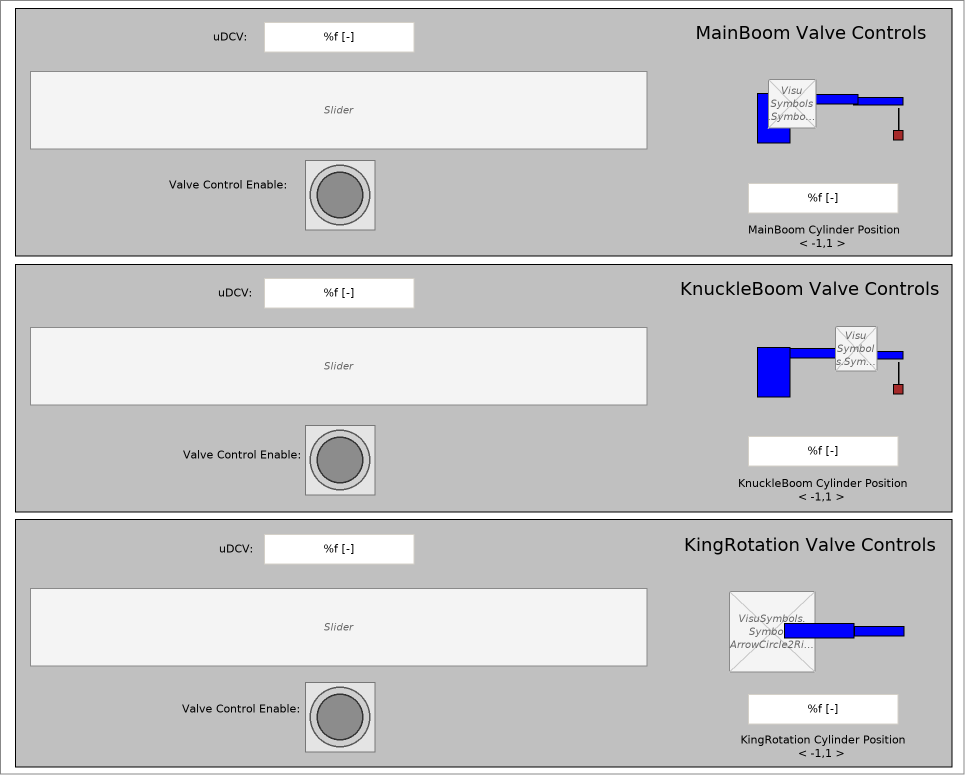
VISUALIZATION Visualization  // 965x775
    RoundedRectangle (15,519 937x248)
    RoundedRectangle (15,264 937x248)
    RoundedRectangle (15,8 937x248)
    Slider (30,71 617x78), variable: Inputs.uDcvMainJib, scale -1..1
    PushSwitchLed (305,160 70x70), variable: Inputs.uDcvEnableMainJib, behaviour: TOGGLE, style: Switch-PushSwitchLed-Gray
    Textfield (264,22 150x30), "%f [-]", text variable: Inputs.uDcvMainJib
        OnMouseClick: write the text variable via Default, min -1, max 1
    Label (197,22 66x30), "uDCV:"
    Label (137,170 182x30), "Valve Control Enable:"
    Slider (30,327 617x78), variable: Inputs.uDcvKnuckleJib, scale -1..1
    PushSwitchLed (305,425 70x70), variable: Inputs.uDcvEnableKnuckleJib, behaviour: TOGGLE, style: Switch-PushSwitchLed-Gray
    Textfield (264,278 150x30), "%f [-]", text variable: Inputs.uDcvKnuckleJib
        OnMouseClick: write the text variable via Default, min -1, max 1
    Label (202,278 66x30), "uDCV:"
    Label (151,440 182x30), "Valve Control Enable:"
    Label (676,18 270x30), "MainBoom Valve Controls"
    Label (675,274 270x30), "KnuckleBoom Valve Controls"
    Slider (30,588 617x78), variable: Inputs.uDcvKingRotation, scale -1..1
    PushSwitchLed (305,682 70x70), variable: Inputs.uDcvEnableKingRotation, behaviour: TOGGLE, style: Switch-PushSwitchLed-Gray
    Textfield (264,534 150x30), "%f [-]", text variable: Inputs.uDcvKingRotation
        OnMouseClick: write the text variable via Default, min -1, max 1
    Label (203,534 66x30), "uDCV:"
    Label (150,694 182x30), "Valve Control Enable:"
    Label (675,530 270x30), "KingRotation Valve Controls"
    Ellipse (757,616 30x30)
    Image (729,591 86x81), angle 320, image: VisuSymbols.Symbols.ArrowCircle2RightRightLeft
    Rectangle (854,626 50x10)
    Rectangle (784,623 70x15)
    Rectangle (887,373 22x1), angle 270
    Rectangle (853,351 50x8), angle 203
    Rectangle (788,348 70x10), angle 349
    Rectangle (757,347 33x50)
    Rectangle (893,384 10x10)
    Rectangle (757,93 33x50)
    Rectangle (887,119 22x1), angle 270
    Rectangle (853,97 50x8), angle 203
    Rectangle (788,94 70x10), angle 349
    Rectangle (893,130 10x10)
    Image (768,79 48x49), angle 345, image: VisuSymbols.Symbols.ArrowCircle2LeftUpDown
    Image (835,326 42x45), angle 10, image: VisuSymbols.Symbols.ArrowCircle2LeftUpDown
    Textfield (748,183 150x30), "%f [-]", text variable: ActuationSystems.fbMainJibCylinderHyd.xPiston
        OnMouseClick: write the text variable via Default, min -1, max 1
    Textfield (748,436 150x30), "%f [-]", text variable: ActuationSystems.fbKnuckleJibCylinderHyd.xPiston
        OnMouseClick: write the text variable via Default, min -1, max 1
    Textfield (748,694 150x30), "%f [-]", text variable: ActuationSystems.fbKingRotationCylinderHyd.xPiston
        OnMouseClick: write the text variable via Default, min -1, max 1
    Label (682,460 282x60), "KnuckleBoom Cylinder Position < -1,1 >"
    Label (682,718 282x57), "KingRotation Cylinder Position < -1,1 >"
    Label (683,206 282x61), "MainBoom Cylinder Position < -1,1 >"
END_VISUALIZATION

(* stored: Version 1.1.0.1, ProductVersion 3.1.4024.9
   Visu Visualization: Id {d8dee94c-064f-4243-8341-9a26801948ea} *)
